{attribute 'enable_dynamic_creation'}
FUNCTION_BLOCK FB_CondiBase
VAR_INPUT
END_VAR
VAR_OUTPUT
END_VAR
VAR_IN_OUT
END_VAR
VAR
	eCondition		: E_Condition;
	pNextCondi		: POINTER TO FB_CondiBase;
	eCondiOperator	: E_LogicOperator;
END_VAR

PROPERTY P_eCondition : E_Condition
SET
eCondition := P_eCondition;
END_SET
END_PROPERTY

METHOD M_ClearNext
VAR_INPUT
END_VAR
IF pNextCondi > 0 THEN
	pNextCondi^.M_ClearNext();
	__DELETE(pNextCondi);
END_IF
END_METHOD

PROPERTY P_eOperator : E_LogicOperator
SET
eCondiOperator := P_eOperator;
END_SET
END_PROPERTY

METHOD M_AddNext
VAR_INPUT
	pCondi : POINTER TO FB_CondiBase;
END_VAR
IF pNextCondi = 0 THEN
	pNextCondi := pCondi;
ELSE
	pNextCondi^.M_AddNext(pCondi);
END_IF
END_METHOD

METHOD M_Check : BYTE
VAR_INPUT
	//bPreResult	: BOOL;
	nPreResult : BYTE;
END_VAR
END_METHOD

END_FUNCTION_BLOCK

(* stored: Version 1.1.0.1, ProductVersion 3.1.4020.12
   POU FB_CondiBase: Id {2a9839b6-9855-4f86-932c-c570a380e71d}, SpecialFunc None
   Property P_eCondition: Id {31d9fe1b-c5cd-479e-bf53-3234e8b3d5b0}
   Set Set: Id {1ce07daf-d2fc-4616-bfd3-e893d0cbd520}
   Method M_ClearNext: Id {4f55be51-86e5-4f49-9aa8-c81e942ea396}
   Property P_eOperator: Id {6e53ba03-9935-4026-aa20-d42cde9cf3c7}
   Set Set: Id {2f4a9737-d101-4cb2-8c79-57b3923ae24f}
   Method M_AddNext: Id {79c20188-50fd-41e8-9b4c-b0b5ddd88bc3}
   Method M_Check: Id {9709da70-775f-4593-8395-0e31a180cd82} *)
